INTERFACE I_AmeClient

END_INTERFACE

(* stored: Version 1.1.0.1, ProductVersion 3.1.4024.12
   Itf I_AmeClient: Id {331a3e02-f3d3-4b18-a5d7-9910e6c08ce3}
   Folder Events: Id {4bfd18d6-0d8b-46e7-abb3-bee0ee031d13} *)
